// TwinCAT 3 PLC project Moving_Average_Filter
// ProgramVersion: 3.1.4024.0
// libraries:
//   Tc2_ControllerToolbox, * (Beckhoff Automation GmbH)
//   Tc2_Standard, * (Beckhoff Automation GmbH)
//   Tc2_System, * (Beckhoff Automation GmbH)
//   Tc3_Module, * (Beckhoff Automation GmbH)
// project tree:
//   / PlcTask.TcTTO
//   POUs/ MAIN.TcPOU, MovingAverageFilter.TcPOU
// real-time tasks:
//   TASK PlcTask: cycle T#10ms, priority 20, ADS port 350

CONFIGURATION Moving_Average_Filter
    RESOURCE PLC ON TwinCAT3
        TASK PlcTask(INTERVAL := T#10ms, PRIORITY := 20);
        PROGRAM MAIN WITH PlcTask : MAIN;
    END_RESOURCE
END_CONFIGURATION

// ---- POUs/MAIN.TcPOU
PROGRAM MAIN
VAR
FBCTRL_MOVING_AVERAGE  :FB_CTRL_MOVING_AVERAGE;
	iejimas: REAL;
	Output: LREAL;
	modas: E_CTRL_MODE;
	ff: ST_CTRL_MOVING_AVERAGE_PARAMS;
	mm: ST_CTRL_NOISE_GENERATOR_PARAMS;
	marius: ARRAY[1..100] OF REAL;
	MovingAverageFilter: MovingAverageFilter;
	FB_CTRL_NOISE_GENERATOR:FB_CTRL_NOISE_GENERATOR;
	adasd: REAL;
	noise: LREAL;
END_VAR

ff.nSamplesToFilter:=5;
ff.tCtrlCycleTime:=T#5H;
ff.tTaskCycleTime:=T#1H;
ff.pWorkArray_ADR:=ADR(marius);
ff.nWorkArray_SIZEOF:=SIZEOF(marius);

mm.fAmplitude:=24;
mm.tCtrlCycleTime:=T#10MS;
mm.tTaskCycleTime:=T#10MS;

FBCTRL_MOVING_AVERAGE(	fIn:=noise ,  	eMode:=ectrl_mode_active, 	fOut=>Output, 	stParams:=ff ); 
MovingAverageFilter(InputValue:=noise, tTaskCycleNumber:=5,SampleNumber:=5,FilterValute=>adasd);
FB_CTRL_NOISE_GENERATOR(fManSyncValue:=12.0,emode:=ectrl_mode_active,Fout=>noise,stParams:=mm);

END_PROGRAM

// ---- POUs/MovingAverageFilter.TcPOU
FUNCTION_BLOCK MovingAverageFilter
VAR_INPUT
	InputValue							:REAL;	
	tTaskCycleNumber					:INT;
	SampleNumber						:INT;
END_VAR
VAR_OUTPUT
	FilterValute						:REAL;
END_VAR
VAR
	i									:INT;	
	MainWorkingArra						:ARRAY[1..10] OF REAL;
	WorkingArraySum						:REAL;
	SumRange							:INT:=0;
	CycleNumber							:INT:=0;
END_VAR

IF tTaskCycleNumber=0 OR tTaskCycleNumber=1 THEN
		    JMP WithoutFilter;
	ELSE
			JMP filter;
END_IF

filter:
	FilterValute:=FilterValueMeth();
//	RETURN;
WithoutFilter:
//	FilterValute:=InputValue;
//	RETURN;

METHOD PRIVATE FilterValueMeth : real
CycleNumber:=CycleNumber+1;
IF CycleNumber=tTaskCycleNumber THEN
	CycleNumber:=0;
	WorkingArraySum:=0;	
	SumRange:=SumRange+1;
	MainWorkingArra[SumRange]:=InputValue;
		FOR i:=1 TO SampleNumber BY 1 DO
			WorkingArraySum:=MainWorkingArra[i]+WorkingArraySum;
		END_FOR	
		IF SumRange=SampleNumber THEN
			SumRange:=0;
		END_IF	
END_IF
FilterValueMeth:=WorkingArraySum/SampleNumber;
END_METHOD

END_FUNCTION_BLOCK
